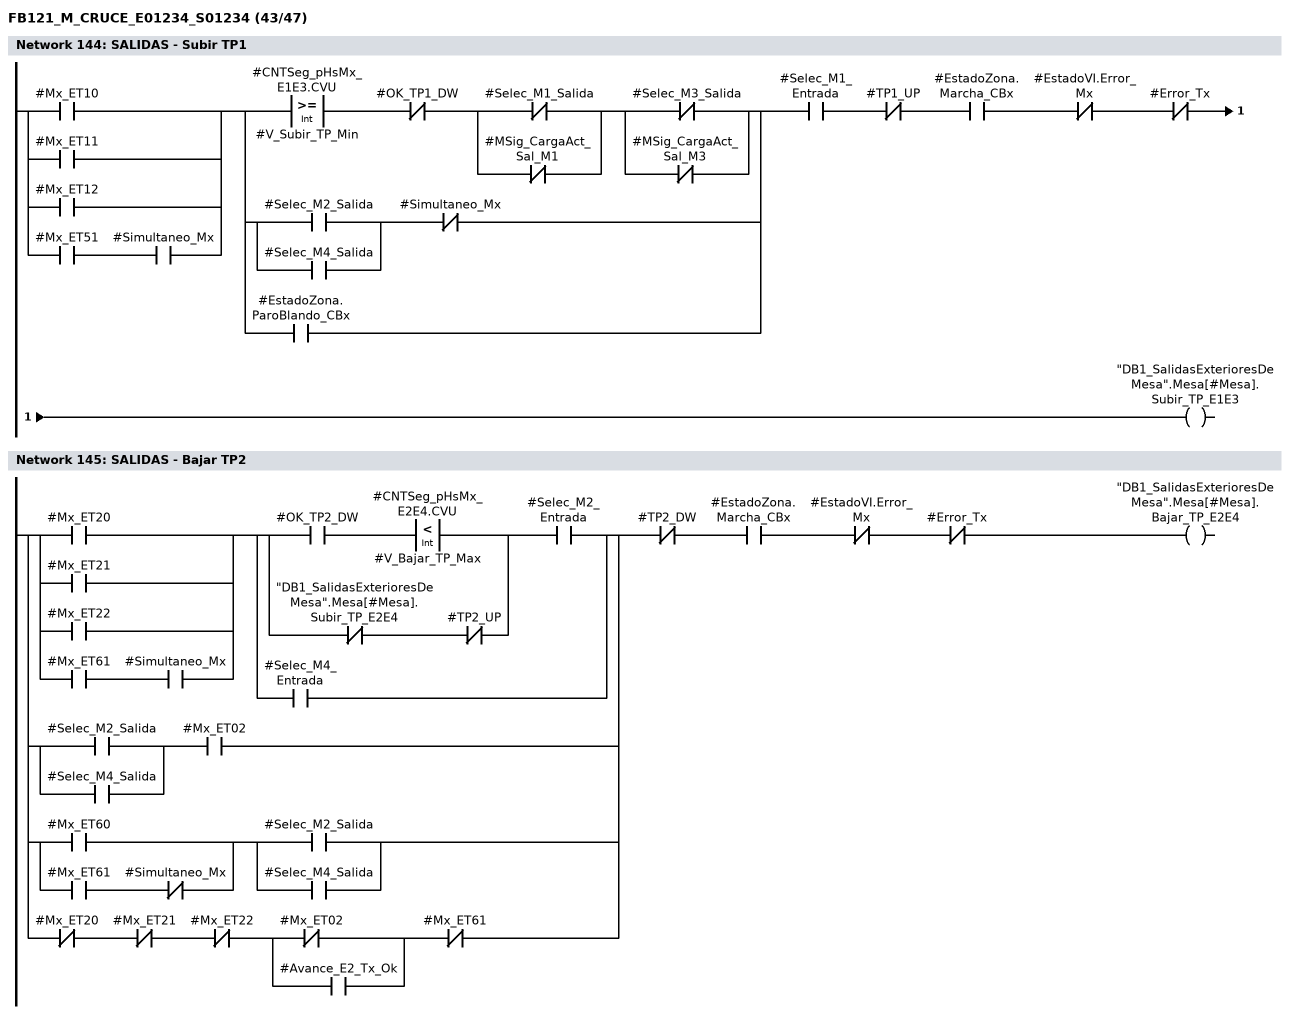
   RUNG wire#powerrail
      Contact( #Mx_ET10 )
      wire#w1
      { S7_Templates := "SrcType := Int" } GE_Contact(in1 := #CNTSeg_pHsMx_E1E3.CVU, in2 := #V_Subir_TP_Min)
      I_Contact( #OK_TP1_DW )
      wire#w2
      I_Contact( #Selec_M1_Salida )
      wire#w3
      I_Contact( #Selec_M3_Salida )
      wire#w4
      Contact( #Selec_M1_Entrada )
      I_Contact( #TP1_UP )
      Contact( #EstadoZona.Marcha_CBx )
      I_Contact( #EstadoVI.Error_Mx )
      I_Contact( #Error_Tx )
      Coil( "DB1_SalidasExterioresDeMesa".Mesa[#Mesa].Subir_TP_E1E3 )
   END_RUNG
   RUNG wire#powerrail
      Contact( #Mx_ET11 )
   END_RUNG wire#w1
   RUNG wire#powerrail
      Contact( #Mx_ET12 )
   END_RUNG wire#w1
   RUNG wire#powerrail
      Contact( #Mx_ET51 )
      Contact( #Simultaneo_Mx )
   END_RUNG wire#w1
   RUNG wire#w2
      I_Contact( #MSig_CargaAct_Sal_M1 )
   END_RUNG wire#w3
   RUNG wire#w3
      I_Contact( #MSig_CargaAct_Sal_M3 )
   END_RUNG wire#w4
   RUNG wire#w1
      Contact( #Selec_M2_Salida )
      wire#w5
      I_Contact( #Simultaneo_Mx )
   END_RUNG wire#w4
   RUNG wire#w1
      Contact( #Selec_M4_Salida )
   END_RUNG wire#w5
   RUNG wire#w1
      Contact( #EstadoZona.ParoBlando_CBx )
   END_RUNG wire#w4
   // the same network as SCL:
   "DB1_SalidasExterioresDeMesa".Mesa[#Mesa].Subir_TP_E1E3 := (#Mx_ET10 OR #Mx_ET11 OR #Mx_ET12 OR (#Mx_ET51 AND #Simultaneo_Mx)) AND (((#CNTSeg_pHsMx_E1E3.CVU >= #V_Subir_TP_Min) AND NOT #OK_TP1_DW AND (NOT #Selec_M1_Salida OR NOT #MSig_CargaAct_Sal_M1) AND (NOT #Selec_M3_Salida OR NOT #MSig_CargaAct_Sal_M3)) OR ((#Selec_M2_Salida OR #Selec_M4_Salida) AND NOT #Simultaneo_Mx) OR #EstadoZona.ParoBlando_CBx) AND #Selec_M1_Entrada AND NOT #TP1_UP AND #EstadoZona.Marcha_CBx AND NOT #EstadoVI.Error_Mx AND NOT #Error_Tx;
END_REGION

REGION Network 145: SALIDAS - Bajar TP2
   RUNG wire#powerrail
      Contact( #Mx_ET20 )
      wire#w1
      Contact( #OK_TP2_DW )
      { S7_Templates := "SrcType := Int" } LT_Contact(in1 := #CNTSeg_pHsMx_E2E4.CVU, in2 := #V_Bajar_TP_Max)
      wire#w2
      Contact( #Selec_M2_Entrada )
      wire#w3
      I_Contact( #TP2_DW )
      Contact( #EstadoZona.Marcha_CBx )
      I_Contact( #EstadoVI.Error_Mx )
      I_Contact( #Error_Tx )
      Coil( "DB1_SalidasExterioresDeMesa".Mesa[#Mesa].Bajar_TP_E2E4 )
   END_RUNG
   RUNG wire#powerrail
      Contact( #Mx_ET21 )
   END_RUNG wire#w1
   RUNG wire#powerrail
      Contact( #Mx_ET22 )
   END_RUNG wire#w1
   RUNG wire#powerrail
      Contact( #Mx_ET61 )
      Contact( #Simultaneo_Mx )
   END_RUNG wire#w1
   RUNG wire#w1
      I_Contact( "DB1_SalidasExterioresDeMesa".Mesa[#Mesa].Subir_TP_E2E4 )
      I_Contact( #TP2_UP )
   END_RUNG wire#w2
   RUNG wire#w1
      Contact( #Selec_M4_Entrada )
   END_RUNG wire#w3
   RUNG wire#powerrail
      Contact( #Selec_M2_Salida )
      wire#w4
      Contact( #Mx_ET02 )
   END_RUNG wire#w3
   RUNG wire#powerrail
      Contact( #Selec_M4_Salida )
   END_RUNG wire#w4
   RUNG wire#powerrail
      Contact( #Mx_ET60 )
      wire#w5
      Contact( #Selec_M2_Salida )
   END_RUNG wire#w3
   RUNG wire#powerrail
      Contact( #Mx_ET61 )
      I_Contact( #Simultaneo_Mx )
   END_RUNG wire#w5
   RUNG wire#w5
      Contact( #Selec_M4_Salida )
   END_RUNG wire#w3
   RUNG wire#powerrail
      I_Contact( #Mx_ET20 )
      I_Contact( #Mx_ET21 )
      I_Contact( #Mx_ET22 )
      wire#w6
      I_Contact( #Mx_ET02 )
      wire#w7
      I_Contact( #Mx_ET61 )
   END_RUNG wire#w3
   RUNG wire#w6
      Contact( #Avance_E2_Tx_Ok )
   END_RUNG wire#w7
   // the same network as SCL:
   "DB1_SalidasExterioresDeMesa".Mesa[#Mesa].Bajar_TP_E2E4 := (((#Mx_ET20 OR #Mx_ET21 OR #Mx_ET22 OR (#Mx_ET61 AND #Simultaneo_Mx)) AND ((((#OK_TP2_DW AND (#CNTSeg_pHsMx_E2E4.CVU < #V_Bajar_TP_Max)) OR (NOT "DB1_SalidasExterioresDeMesa".Mesa[#Mesa].Subir_TP_E2E4 AND NOT #TP2_UP)) AND #Selec_M2_Entrada) OR #Selec_M4_Entrada)) OR ((#Selec_M2_Salida OR #Selec_M4_Salida) AND #Mx_ET02) OR ((#Mx_ET60 OR (#Mx_ET61 AND NOT #Simultaneo_Mx)) AND (#Selec_M2_Salida OR #Selec_M4_Salida)) OR (NOT #Mx_ET20 AND NOT #Mx_ET21 AND NOT #Mx_ET22 AND (NOT #Mx_ET02 OR #Avance_E2_Tx_Ok) AND NOT #Mx_ET61)) AND NOT #TP2_DW AND #EstadoZona.Marcha_CBx AND NOT #EstadoVI.Error_Mx AND NOT #Error_Tx;
END_REGION

REGION Network 146: SALIDAS - Subir TP2
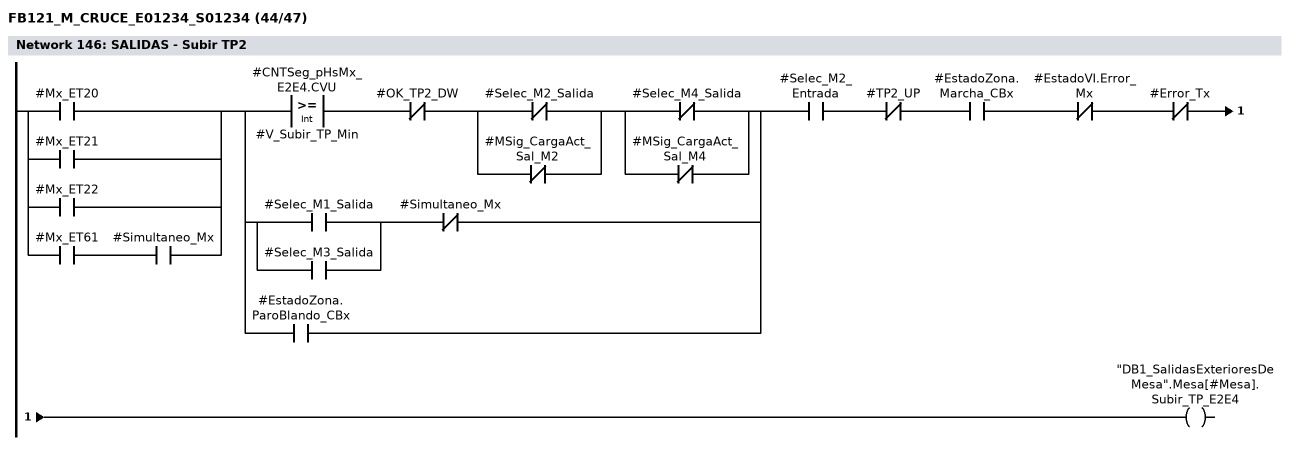
   RUNG wire#powerrail
      Contact( #Mx_ET20 )
      wire#w1
      { S7_Templates := "SrcType := Int" } GE_Contact(in1 := #CNTSeg_pHsMx_E2E4.CVU, in2 := #V_Subir_TP_Min)
      I_Contact( #OK_TP2_DW )
      wire#w2
      I_Contact( #Selec_M2_Salida )
      wire#w3
      I_Contact( #Selec_M4_Salida )
      wire#w4
      Contact( #Selec_M2_Entrada )
      I_Contact( #TP2_UP )
      Contact( #EstadoZona.Marcha_CBx )
      I_Contact( #EstadoVI.Error_Mx )
      I_Contact( #Error_Tx )
      Coil( "DB1_SalidasExterioresDeMesa".Mesa[#Mesa].Subir_TP_E2E4 )
   END_RUNG
   RUNG wire#powerrail
      Contact( #Mx_ET21 )
   END_RUNG wire#w1
   RUNG wire#powerrail
      Contact( #Mx_ET22 )
   END_RUNG wire#w1
   RUNG wire#powerrail
      Contact( #Mx_ET61 )
      Contact( #Simultaneo_Mx )
   END_RUNG wire#w1
   RUNG wire#w2
      I_Contact( #MSig_CargaAct_Sal_M2 )
   END_RUNG wire#w3
   RUNG wire#w3
      I_Contact( #MSig_CargaAct_Sal_M4 )
   END_RUNG wire#w4
   RUNG wire#w1
      Contact( #Selec_M1_Salida )
      wire#w5
      I_Contact( #Simultaneo_Mx )
   END_RUNG wire#w4
   RUNG wire#w1
      Contact( #Selec_M3_Salida )
   END_RUNG wire#w5
   RUNG wire#w1
      Contact( #EstadoZona.ParoBlando_CBx )
   END_RUNG wire#w4
   // the same network as SCL:
   "DB1_SalidasExterioresDeMesa".Mesa[#Mesa].Subir_TP_E2E4 := (#Mx_ET20 OR #Mx_ET21 OR #Mx_ET22 OR (#Mx_ET61 AND #Simultaneo_Mx)) AND (((#CNTSeg_pHsMx_E2E4.CVU >= #V_Subir_TP_Min) AND NOT #OK_TP2_DW AND (NOT #Selec_M2_Salida OR NOT #MSig_CargaAct_Sal_M2) AND (NOT #Selec_M4_Salida OR NOT #MSig_CargaAct_Sal_M4)) OR ((#Selec_M1_Salida OR #Selec_M3_Salida) AND NOT #Simultaneo_Mx) OR #EstadoZona.ParoBlando_CBx) AND #Selec_M2_Entrada AND NOT #TP2_UP AND #EstadoZona.Marcha_CBx AND NOT #EstadoVI.Error_Mx AND NOT #Error_Tx;
END_REGION

REGION Network 147: ESTADOS DE LA MESA
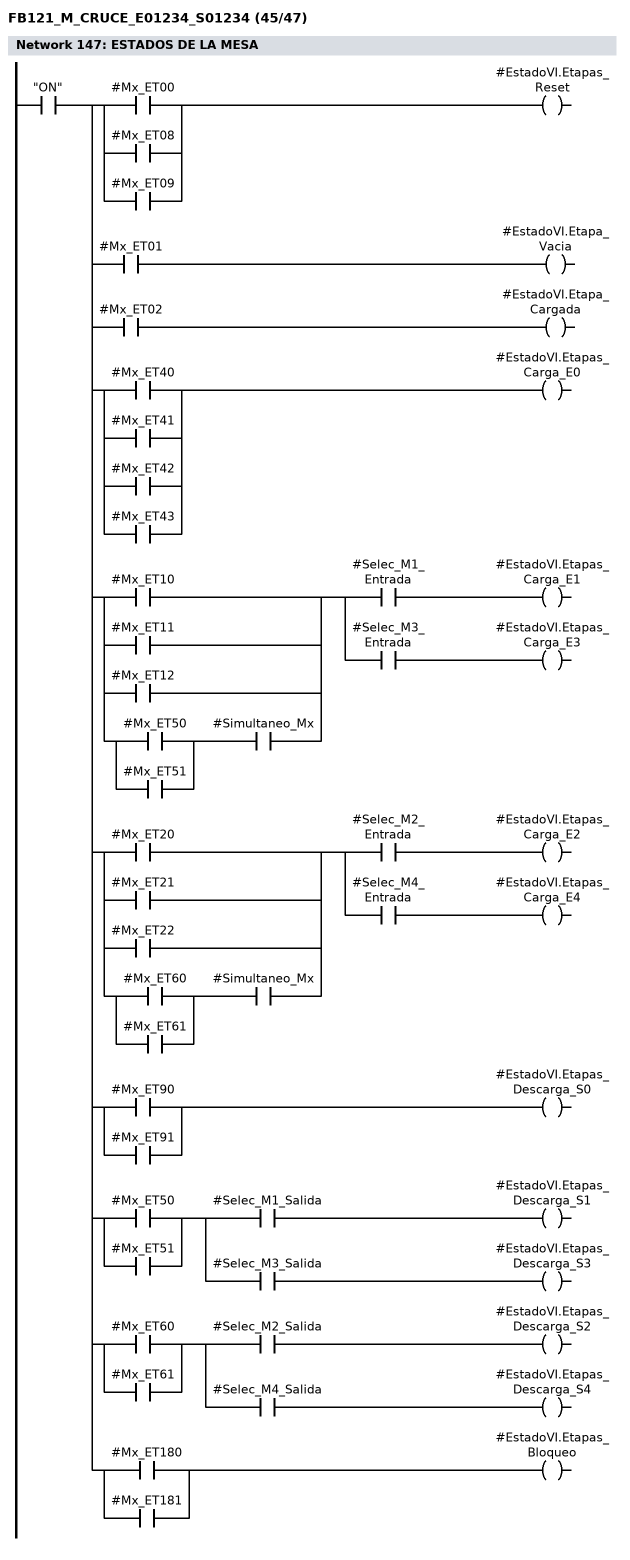
   RUNG wire#powerrail
      Contact( "ON" )
      wire#w1
      Contact( #Mx_ET00 )
      wire#w2
      Coil( #EstadoVI.Etapas_Reset )
   END_RUNG
   RUNG wire#w1
      Contact( #Mx_ET08 )
   END_RUNG wire#w2
   RUNG wire#w1
      Contact( #Mx_ET09 )
   END_RUNG wire#w2
   RUNG wire#w1
      Contact( #Mx_ET01 )
      Coil( #EstadoVI.Etapa_Vacia )
   END_RUNG
   RUNG wire#w1
      Contact( #Mx_ET02 )
      Coil( #EstadoVI.Etapa_Cargada )
   END_RUNG
   RUNG wire#w1
      Contact( #Mx_ET40 )
      wire#w3
      Coil( #EstadoVI.Etapas_Carga_E0 )
   END_RUNG
   RUNG wire#w1
      Contact( #Mx_ET41 )
   END_RUNG wire#w3
   RUNG wire#w1
      Contact( #Mx_ET42 )
   END_RUNG wire#w3
   RUNG wire#w1
      Contact( #Mx_ET43 )
   END_RUNG wire#w3
   RUNG wire#w1
      Contact( #Mx_ET10 )
      wire#w4
      Contact( #Selec_M1_Entrada )
      Coil( #EstadoVI.Etapas_Carga_E1 )
   END_RUNG
   RUNG wire#w1
      Contact( #Mx_ET11 )
   END_RUNG wire#w4
   RUNG wire#w1
      Contact( #Mx_ET12 )
   END_RUNG wire#w4
   RUNG wire#w1
      Contact( #Mx_ET50 )
      wire#w5
      Contact( #Simultaneo_Mx )
   END_RUNG wire#w4
   RUNG wire#w1
      Contact( #Mx_ET51 )
   END_RUNG wire#w5
   RUNG wire#w4
      Contact( #Selec_M3_Entrada )
      Coil( #EstadoVI.Etapas_Carga_E3 )
   END_RUNG
   RUNG wire#w1
      Contact( #Mx_ET20 )
      wire#w6
      Contact( #Selec_M2_Entrada )
      Coil( #EstadoVI.Etapas_Carga_E2 )
   END_RUNG
   RUNG wire#w1
      Contact( #Mx_ET21 )
   END_RUNG wire#w6
   RUNG wire#w1
      Contact( #Mx_ET22 )
   END_RUNG wire#w6
   RUNG wire#w1
      Contact( #Mx_ET60 )
      wire#w7
      Contact( #Simultaneo_Mx )
   END_RUNG wire#w6
   RUNG wire#w1
      Contact( #Mx_ET61 )
   END_RUNG wire#w7
   RUNG wire#w6
      Contact( #Selec_M4_Entrada )
      Coil( #EstadoVI.Etapas_Carga_E4 )
   END_RUNG
   RUNG wire#w1
      Contact( #Mx_ET90 )
      wire#w8
      Coil( #EstadoVI.Etapas_Descarga_S0 )
   END_RUNG
   RUNG wire#w1
      Contact( #Mx_ET91 )
   END_RUNG wire#w8
   RUNG wire#w1
      Contact( #Mx_ET50 )
      wire#w9
      Contact( #Selec_M1_Salida )
      Coil( #EstadoVI.Etapas_Descarga_S1 )
   END_RUNG
   RUNG wire#w1
      Contact( #Mx_ET51 )
   END_RUNG wire#w9
   RUNG wire#w9
      Contact( #Selec_M3_Salida )
      Coil( #EstadoVI.Etapas_Descarga_S3 )
   END_RUNG
   RUNG wire#w1
      Contact( #Mx_ET60 )
      wire#w10
      Contact( #Selec_M2_Salida )
      Coil( #EstadoVI.Etapas_Descarga_S2 )
   END_RUNG
   RUNG wire#w1
      Contact( #Mx_ET61 )
   END_RUNG wire#w10
   RUNG wire#w10
      Contact( #Selec_M4_Salida )
      Coil( #EstadoVI.Etapas_Descarga_S4 )
   END_RUNG
   RUNG wire#w1
      Contact( #Mx_ET180 )
      wire#w11
      Coil( #EstadoVI.Etapas_Bloqueo )
   END_RUNG
   RUNG wire#w1
      Contact( #Mx_ET181 )
   END_RUNG wire#w11
   // the same network as SCL:
   #EstadoVI.Etapas_Reset := "ON" AND (#Mx_ET00 OR #Mx_ET08 OR #Mx_ET09);
   #EstadoVI.Etapa_Vacia := "ON" AND #Mx_ET01;
   #EstadoVI.Etapa_Cargada := "ON" AND #Mx_ET02;
   #EstadoVI.Etapas_Carga_E0 := "ON" AND (#Mx_ET40 OR #Mx_ET41 OR #Mx_ET42 OR #Mx_ET43);
   #_w1 := "ON" AND (#Mx_ET10 OR #Mx_ET11 OR #Mx_ET12 OR ((#Mx_ET50 OR #Mx_ET51) AND #Simultaneo_Mx));
   #EstadoVI.Etapas_Carga_E1 := #_w1 AND #Selec_M1_Entrada;
   #EstadoVI.Etapas_Carga_E3 := #_w1 AND #Selec_M3_Entrada;
   #_w2 := "ON" AND (#Mx_ET20 OR #Mx_ET21 OR #Mx_ET22 OR ((#Mx_ET60 OR #Mx_ET61) AND #Simultaneo_Mx));
   #EstadoVI.Etapas_Carga_E2 := #_w2 AND #Selec_M2_Entrada;
   #EstadoVI.Etapas_Carga_E4 := #_w2 AND #Selec_M4_Entrada;
   #EstadoVI.Etapas_Descarga_S0 := "ON" AND (#Mx_ET90 OR #Mx_ET91);
   #_w3 := "ON" AND (#Mx_ET50 OR #Mx_ET51);
   #EstadoVI.Etapas_Descarga_S1 := #_w3 AND #Selec_M1_Salida;
   #EstadoVI.Etapas_Descarga_S3 := #_w3 AND #Selec_M3_Salida;
   #_w4 := "ON" AND (#Mx_ET60 OR #Mx_ET61);
   #EstadoVI.Etapas_Descarga_S2 := #_w4 AND #Selec_M2_Salida;
   #EstadoVI.Etapas_Descarga_S4 := #_w4 AND #Selec_M4_Salida;
   #EstadoVI.Etapas_Bloqueo := "ON" AND (#Mx_ET180 OR #Mx_ET181);
END_REGION

REGION Network 148: ESTADO ENTRADAS DE LA MESA
   // MODIF: TRANSFER UP, TRANSFER_DW, TOPE_UP_2, TOPE_DW_2
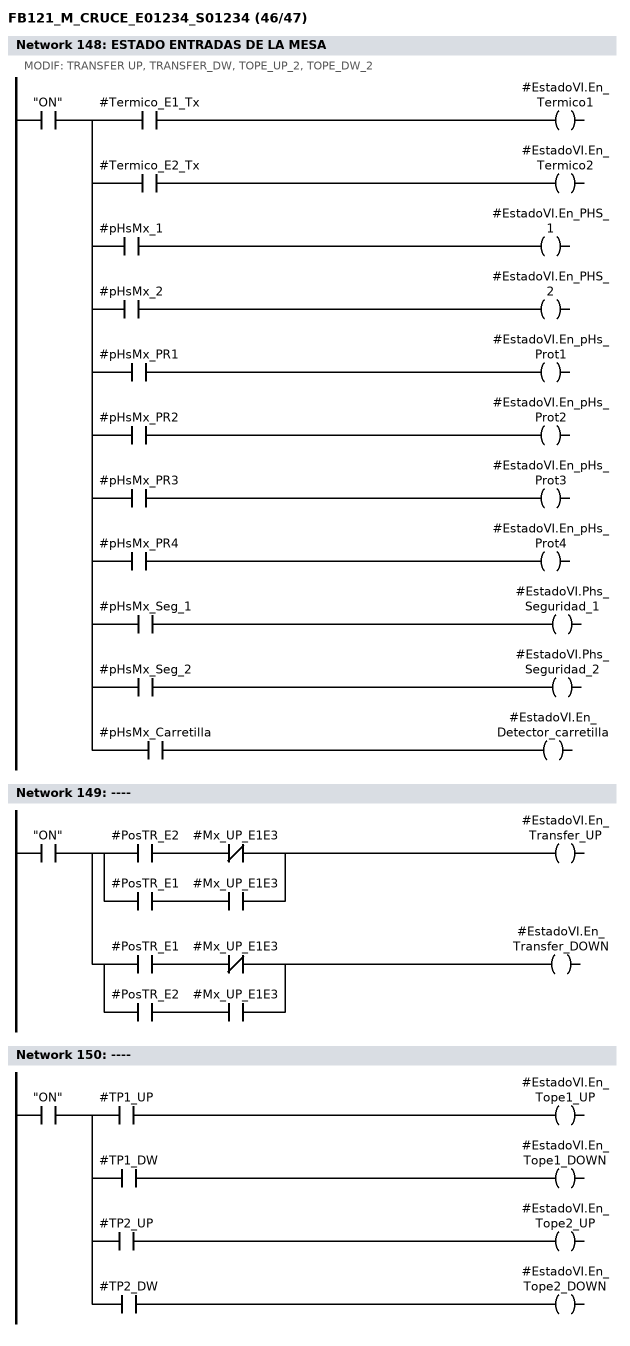
   RUNG wire#powerrail
      Contact( "ON" )
      wire#w1
      Contact( #Termico_E1_Tx )
      Coil( #EstadoVI.En_Termico1 )
   END_RUNG
   RUNG wire#w1
      Contact( #Termico_E2_Tx )
      Coil( #EstadoVI.En_Termico2 )
   END_RUNG
   RUNG wire#w1
      Contact( #pHsMx_1 )
      Coil( #EstadoVI.En_PHS_1 )
   END_RUNG
   RUNG wire#w1
      Contact( #pHsMx_2 )
      Coil( #EstadoVI.En_PHS_2 )
   END_RUNG
   RUNG wire#w1
      Contact( #pHsMx_PR1 )
      Coil( #EstadoVI.En_pHs_Prot1 )
   END_RUNG
   RUNG wire#w1
      Contact( #pHsMx_PR2 )
      Coil( #EstadoVI.En_pHs_Prot2 )
   END_RUNG
   RUNG wire#w1
      Contact( #pHsMx_PR3 )
      Coil( #EstadoVI.En_pHs_Prot3 )
   END_RUNG
   RUNG wire#w1
      Contact( #pHsMx_PR4 )
      Coil( #EstadoVI.En_pHs_Prot4 )
   END_RUNG
   RUNG wire#w1
      Contact( #pHsMx_Seg_1 )
      Coil( #EstadoVI.Phs_Seguridad_1 )
   END_RUNG
   RUNG wire#w1
      Contact( #pHsMx_Seg_2 )
      Coil( #EstadoVI.Phs_Seguridad_2 )
   END_RUNG
   RUNG wire#w1
      Contact( #pHsMx_Carretilla )
      Coil( #EstadoVI.En_Detector_carretilla )
   END_RUNG
   // the same network as SCL:
   #EstadoVI.En_Termico1 := "ON" AND #Termico_E1_Tx;
   #EstadoVI.En_Termico2 := "ON" AND #Termico_E2_Tx;
   #EstadoVI.En_PHS_1 := "ON" AND #pHsMx_1;
   #EstadoVI.En_PHS_2 := "ON" AND #pHsMx_2;
   #EstadoVI.En_pHs_Prot1 := "ON" AND #pHsMx_PR1;
   #EstadoVI.En_pHs_Prot2 := "ON" AND #pHsMx_PR2;
   #EstadoVI.En_pHs_Prot3 := "ON" AND #pHsMx_PR3;
   #EstadoVI.En_pHs_Prot4 := "ON" AND #pHsMx_PR4;
   #EstadoVI.Phs_Seguridad_1 := "ON" AND #pHsMx_Seg_1;
   #EstadoVI.Phs_Seguridad_2 := "ON" AND #pHsMx_Seg_2;
   #EstadoVI.En_Detector_carretilla := "ON" AND #pHsMx_Carretilla;
END_REGION

REGION Network 149: ----
   RUNG wire#powerrail
      Contact( "ON" )
      wire#w1
      Contact( #PosTR_E2 )
      I_Contact( #Mx_UP_E1E3 )
      wire#w2
      Coil( #EstadoVI.En_Transfer_UP )
   END_RUNG
   RUNG wire#w1
      Contact( #PosTR_E1 )
      Contact( #Mx_UP_E1E3 )
   END_RUNG wire#w2
   RUNG wire#w1
      Contact( #PosTR_E1 )
      I_Contact( #Mx_UP_E1E3 )
      wire#w3
      Coil( #EstadoVI.En_Transfer_DOWN )
   END_RUNG
   RUNG wire#w1
      Contact( #PosTR_E2 )
      Contact( #Mx_UP_E1E3 )
   END_RUNG wire#w3
   // the same network as SCL:
   #EstadoVI.En_Transfer_UP := "ON" AND ((#PosTR_E2 AND NOT #Mx_UP_E1E3) OR (#PosTR_E1 AND #Mx_UP_E1E3));
   #EstadoVI.En_Transfer_DOWN := "ON" AND ((#PosTR_E1 AND NOT #Mx_UP_E1E3) OR (#PosTR_E2 AND #Mx_UP_E1E3));
END_REGION

REGION Network 150: ----
   RUNG wire#powerrail
      Contact( "ON" )
      wire#w1
      Contact( #TP1_UP )
      Coil( #EstadoVI.En_Tope1_UP )
   END_RUNG
   RUNG wire#w1
      Contact( #TP1_DW )
      Coil( #EstadoVI.En_Tope1_DOWN )
   END_RUNG
   RUNG wire#w1
      Contact( #TP2_UP )
      Coil( #EstadoVI.En_Tope2_UP )
   END_RUNG
   RUNG wire#w1
      Contact( #TP2_DW )
      Coil( #EstadoVI.En_Tope2_DOWN )
   END_RUNG
   // the same network as SCL:
   #EstadoVI.En_Tope1_UP := "ON" AND #TP1_UP;
   #EstadoVI.En_Tope1_DOWN := "ON" AND #TP1_DW;
   #EstadoVI.En_Tope2_UP := "ON" AND #TP2_UP;
   #EstadoVI.En_Tope2_DOWN := "ON" AND #TP2_DW;
END_REGION

REGION Network 151: SALIDAS DE LA MESA
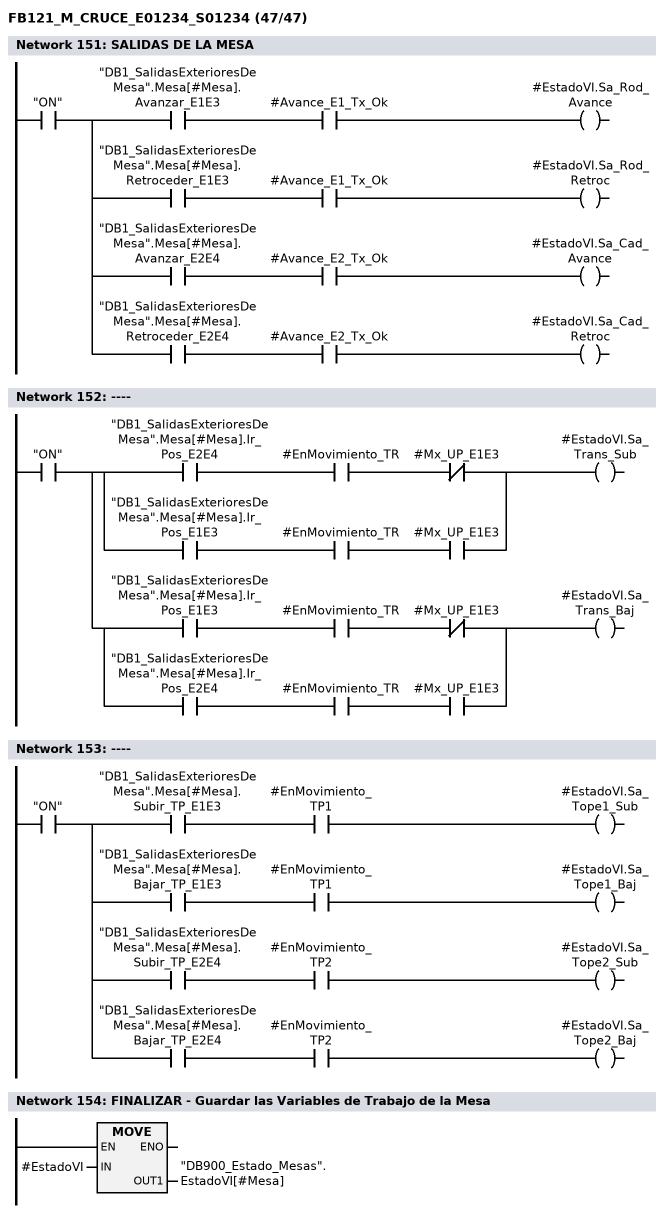
   RUNG wire#powerrail
      Contact( "ON" )
      wire#w1
      Contact( "DB1_SalidasExterioresDeMesa".Mesa[#Mesa].Avanzar_E1E3 )
      Contact( #Avance_E1_Tx_Ok )
      Coil( #EstadoVI.Sa_Rod_Avance )
   END_RUNG
   RUNG wire#w1
      Contact( "DB1_SalidasExterioresDeMesa".Mesa[#Mesa].Retroceder_E1E3 )
      Contact( #Avance_E1_Tx_Ok )
      Coil( #EstadoVI.Sa_Rod_Retroc )
   END_RUNG
   RUNG wire#w1
      Contact( "DB1_SalidasExterioresDeMesa".Mesa[#Mesa].Avanzar_E2E4 )
      Contact( #Avance_E2_Tx_Ok )
      Coil( #EstadoVI.Sa_Cad_Avance )
   END_RUNG
   RUNG wire#w1
      Contact( "DB1_SalidasExterioresDeMesa".Mesa[#Mesa].Retroceder_E2E4 )
      Contact( #Avance_E2_Tx_Ok )
      Coil( #EstadoVI.Sa_Cad_Retroc )
   END_RUNG
   // the same network as SCL:
   #EstadoVI.Sa_Rod_Avance := "ON" AND "DB1_SalidasExterioresDeMesa".Mesa[#Mesa].Avanzar_E1E3 AND #Avance_E1_Tx_Ok;
   #EstadoVI.Sa_Rod_Retroc := "ON" AND "DB1_SalidasExterioresDeMesa".Mesa[#Mesa].Retroceder_E1E3 AND #Avance_E1_Tx_Ok;
   #EstadoVI.Sa_Cad_Avance := "ON" AND "DB1_SalidasExterioresDeMesa".Mesa[#Mesa].Avanzar_E2E4 AND #Avance_E2_Tx_Ok;
   #EstadoVI.Sa_Cad_Retroc := "ON" AND "DB1_SalidasExterioresDeMesa".Mesa[#Mesa].Retroceder_E2E4 AND #Avance_E2_Tx_Ok;
END_REGION

REGION Network 152: ----
   RUNG wire#powerrail
      Contact( "ON" )
      wire#w1
      Contact( "DB1_SalidasExterioresDeMesa".Mesa[#Mesa].Ir_Pos_E2E4 )
      Contact( #EnMovimiento_TR )
      I_Contact( #Mx_UP_E1E3 )
      wire#w2
      Coil( #EstadoVI.Sa_Trans_Sub )
   END_RUNG
   RUNG wire#w1
      Contact( "DB1_SalidasExterioresDeMesa".Mesa[#Mesa].Ir_Pos_E1E3 )
      Contact( #EnMovimiento_TR )
      Contact( #Mx_UP_E1E3 )
   END_RUNG wire#w2
   RUNG wire#w1
      Contact( "DB1_SalidasExterioresDeMesa".Mesa[#Mesa].Ir_Pos_E1E3 )
      Contact( #EnMovimiento_TR )
      I_Contact( #Mx_UP_E1E3 )
      wire#w3
      Coil( #EstadoVI.Sa_Trans_Baj )
   END_RUNG
   RUNG wire#w1
      Contact( "DB1_SalidasExterioresDeMesa".Mesa[#Mesa].Ir_Pos_E2E4 )
      Contact( #EnMovimiento_TR )
      Contact( #Mx_UP_E1E3 )
   END_RUNG wire#w3
   // the same network as SCL:
   #EstadoVI.Sa_Trans_Sub := "ON" AND (("DB1_SalidasExterioresDeMesa".Mesa[#Mesa].Ir_Pos_E2E4 AND #EnMovimiento_TR AND NOT #Mx_UP_E1E3) OR ("DB1_SalidasExterioresDeMesa".Mesa[#Mesa].Ir_Pos_E1E3 AND #EnMovimiento_TR AND #Mx_UP_E1E3));
   #EstadoVI.Sa_Trans_Baj := "ON" AND (("DB1_SalidasExterioresDeMesa".Mesa[#Mesa].Ir_Pos_E1E3 AND #EnMovimiento_TR AND NOT #Mx_UP_E1E3) OR ("DB1_SalidasExterioresDeMesa".Mesa[#Mesa].Ir_Pos_E2E4 AND #EnMovimiento_TR AND #Mx_UP_E1E3));
END_REGION

REGION Network 153: ----
   RUNG wire#powerrail
      Contact( "ON" )
      wire#w1
      Contact( "DB1_SalidasExterioresDeMesa".Mesa[#Mesa].Subir_TP_E1E3 )
      Contact( #EnMovimiento_TP1 )
      Coil( #EstadoVI.Sa_Tope1_Sub )
   END_RUNG
   RUNG wire#w1
      Contact( "DB1_SalidasExterioresDeMesa".Mesa[#Mesa].Bajar_TP_E1E3 )
      Contact( #EnMovimiento_TP1 )
      Coil( #EstadoVI.Sa_Tope1_Baj )
   END_RUNG
   RUNG wire#w1
      Contact( "DB1_SalidasExterioresDeMesa".Mesa[#Mesa].Subir_TP_E2E4 )
      Contact( #EnMovimiento_TP2 )
      Coil( #EstadoVI.Sa_Tope2_Sub )
   END_RUNG
   RUNG wire#w1
      Contact( "DB1_SalidasExterioresDeMesa".Mesa[#Mesa].Bajar_TP_E2E4 )
      Contact( #EnMovimiento_TP2 )
      Coil( #EstadoVI.Sa_Tope2_Baj )
   END_RUNG
   // the same network as SCL:
   #EstadoVI.Sa_Tope1_Sub := "ON" AND "DB1_SalidasExterioresDeMesa".Mesa[#Mesa].Subir_TP_E1E3 AND #EnMovimiento_TP1;
   #EstadoVI.Sa_Tope1_Baj := "ON" AND "DB1_SalidasExterioresDeMesa".Mesa[#Mesa].Bajar_TP_E1E3 AND #EnMovimiento_TP1;
   #EstadoVI.Sa_Tope2_Sub := "ON" AND "DB1_SalidasExterioresDeMesa".Mesa[#Mesa].Subir_TP_E2E4 AND #EnMovimiento_TP2;
   #EstadoVI.Sa_Tope2_Baj := "ON" AND "DB1_SalidasExterioresDeMesa".Mesa[#Mesa].Bajar_TP_E2E4 AND #EnMovimiento_TP2;
END_REGION

REGION Network 154: FINALIZAR - Guardar las Variables de Trabajo de la Mesa
   RUNG wire#powerrail
      Move(in := #EstadoVI, out1 => "DB900_Estado_Mesas".EstadoVI[#Mesa])
   END_RUNG
   // the same network as SCL:
   "DB900_Estado_Mesas".EstadoVI[#Mesa] := #EstadoVI;
END_REGION
END_FUNCTION_BLOCK
